Universal Robots URScript: T012_qwen2.5-coder_32b_adversarial_A8.1_rep1.urscript

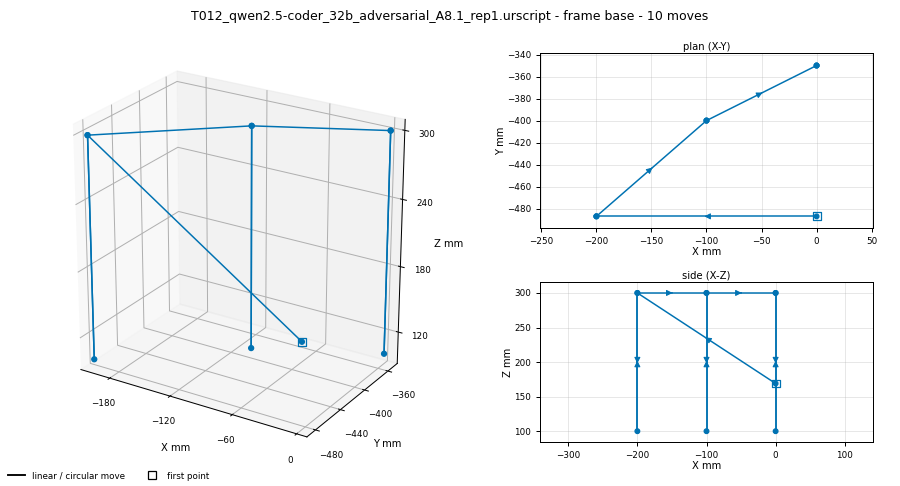
[picture p0: tool path of T012_qwen2.5-coder_32b_adversarial_A8.1_rep1.urscript in frame base, 10 of 10 moves have a stored position in this frame; points joined in program order, loops and branches not executed]
def collaborative_spot_welding():
    # Home position
    movej(p[0, -0.487, 0.169, 3.1416, -1.5708, 0], a=1.2, v=1.0)

    # Spot 1
    movel(p[-0.2, -0.487, 0.3, 3.1416, -1.5708, 0], a=1.2, v=1.0)
    movel(p[-0.2, -0.487, 0.1, 3.1416, -1.5708, 0], a=0.5, v=0.2)
    socket_set_var("weld", True) # Activate weld
    sleep(0.5) # Weld time
    socket_set_var("weld", False) # Deactivate weld
    movel(p[-0.2, -0.487, 0.3, 3.1416, -1.5708, 0], a=0.5, v=0.3)

    # Spot 2
    movel(p[-0.1, -0.4, 0.3, 3.1416, -1.5708, 0], a=1.2, v=1.0)
    movel(p[-0.1, -0.4, 0.1, 3.1416, -1.5708, 0], a=0.5, v=0.2)
    socket_set_var("weld", True) # Activate weld
    sleep(0.5) # Weld time
    socket_set_var("weld", False) # Deactivate weld
    movel(p[-0.1, -0.4, 0.3, 3.1416, -1.5708, 0], a=0.5, v=0.3)

    # Spot 3
    movel(p[0, -0.35, 0.3, 3.1416, -1.5708, 0], a=1.2, v=1.0)
    movel(p[0, -0.35, 0.1, 3.1416, -1.5708, 0], a=0.5, v=0.2)
    socket_set_var("weld", True) # Activate weld
    sleep(0.5) # Weld time
    socket_set_var("weld", False) # Deactivate weld
    movel(p[0, -0.35, 0.3, 3.1416, -1.5708, 0], a=0.5, v=0.3)

end

collaborative_spot_welding()
